Universal Robots PolyScope program: Aufgabe1_2.urp

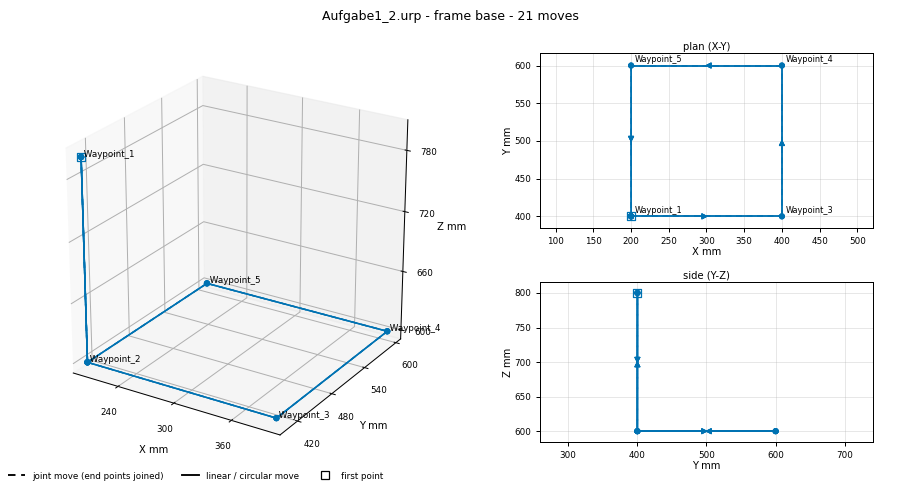
[picture p0: tool path of Aufgabe1_2.urp in frame base, 21 of 21 moves have a stored position in this frame; points joined in program order, loops and branches not executed]
Program Aufgabe1_2 (installation=default directory=/home/ur/ursim-current/programs/new folder createdIn=5.12.4.1101661 lastSavedIn=5.12.4.1101661 robotSerialNumber=20195599999)
Calibrated DH parameters: a=[0, -0.425, -0.3922, 0, 0, 0]; d=[0.1625, 0, 0, 0.1333, 0.0997, 0.0996]; alpha=[1.570796, 0, 0, 1.570796, -1.570796, 0]; deltaTheta=[0, 0, 0, 0, 0, 0]
Robot Program (runOnlyOnce=false)
  MoveL speed 250 mm/s, acceleration 1200 mm/s^2 (useActiveTCP=true) feature=Base
    Waypoint Waypoint_1: TCP in base x=200.031 y=400.097 z=800.02 mm, rx=0 ry=3.1204 rz=0 rad; joints [-133.696, -75.689, 20.033, -35.183, 269.122, 136.298] deg
    MoveL speed 250 mm/s, acceleration 1200 mm/s^2 (useActiveTCP=true) feature=Base
      Waypoint Waypoint_2: TCP in base x=200.014 y=400.002 z=600.007 mm, rx=0 ry=3.1204 rz=0 rad; joints [-133.703, -96.648, 79.829, -74.02, 269.122, 136.29] deg
      Waypoint Waypoint_3: TCP in base x=400.007 y=400.002 z=600.007 mm, rx=0 ry=3.1204 rz=0 rad; joints [-148.515, -79.953, 62.627, -73.709, 269.366, 121.479] deg
      Waypoint Waypoint_4: TCP in base x=400.007 y=600.024 z=600.007 mm, rx=0 ry=3.1204 rz=0 rad; joints [-134.219, -48.622, 15.08, -57.305, 269.13, 135.774] deg
      Waypoint Waypoint_5: TCP in base x=200.031 y=600.024 z=600.007 mm, rx=0 ry=3.1204 rz=0 rad; joints [-120.435, -69.177, 48.455, -69.893, 268.953, 149.559] deg
      Waypoint Waypoint_2: TCP in base x=200.014 y=400.002 z=600.007 mm, rx=0 ry=3.1204 rz=0 rad; joints [-133.703, -96.648, 79.829, -74.02, 269.122, 136.29] deg
      MoveL speed 250 mm/s, acceleration 1200 mm/s^2 (useActiveTCP=true) feature=Base
        Waypoint Waypoint_1: TCP in base x=200.031 y=400.097 z=800.02 mm, rx=0 ry=3.1204 rz=0 rad; joints [-133.696, -75.689, 20.033, -35.183, 269.122, 136.298] deg
  MoveJ speed 60 deg/s, acceleration 80 deg/s^2 (useActiveTCP=true) feature=Base
    Waypoint Waypoint_1: TCP in base x=200.031 y=400.097 z=800.02 mm, rx=0 ry=3.1204 rz=0 rad; joints [-133.696, -75.689, 20.033, -35.183, 269.122, 136.298] deg
    MoveJ speed 60 deg/s, acceleration 80 deg/s^2 (useActiveTCP=true) feature=Base
      Waypoint Waypoint_2: TCP in base x=200.014 y=400.002 z=600.007 mm, rx=0 ry=3.1204 rz=0 rad; joints [-133.703, -96.648, 79.829, -74.02, 269.122, 136.29] deg
      Waypoint Waypoint_3: TCP in base x=400.007 y=400.002 z=600.007 mm, rx=0 ry=3.1204 rz=0 rad; joints [-148.515, -79.953, 62.627, -73.709, 269.366, 121.479] deg
      Waypoint Waypoint_4: TCP in base x=400.007 y=600.024 z=600.007 mm, rx=0 ry=3.1204 rz=0 rad; joints [-134.219, -48.622, 15.08, -57.305, 269.13, 135.774] deg
      Waypoint Waypoint_5: TCP in base x=200.031 y=600.024 z=600.007 mm, rx=0 ry=3.1204 rz=0 rad; joints [-120.435, -69.177, 48.455, -69.893, 268.953, 149.559] deg
      Waypoint Waypoint_2: TCP in base x=200.014 y=400.002 z=600.007 mm, rx=0 ry=3.1204 rz=0 rad; joints [-133.703, -96.648, 79.829, -74.02, 269.122, 136.29] deg
      MoveJ speed 60 deg/s, acceleration 80 deg/s^2 (useActiveTCP=true) feature=Base
        Waypoint Waypoint_1: TCP in base x=200.031 y=400.097 z=800.02 mm, rx=0 ry=3.1204 rz=0 rad; joints [-133.696, -75.689, 20.033, -35.183, 269.122, 136.298] deg
  MoveP speed 250 mm/s, acceleration 1200 mm/s^2 (blendRadius=0.025 useActiveTCP=true) feature=Base
    Waypoint Waypoint_1: TCP in base x=200.031 y=400.097 z=800.02 mm, rx=0 ry=3.1204 rz=0 rad; joints [-133.696, -75.689, 20.033, -35.183, 269.122, 136.298] deg
    MoveP speed 250 mm/s, acceleration 1200 mm/s^2 (blendRadius=0.025 useActiveTCP=true) feature=Base
      Waypoint Waypoint_2: TCP in base x=200.014 y=400.002 z=600.007 mm, rx=0 ry=3.1204 rz=0 rad; joints [-133.703, -96.648, 79.829, -74.02, 269.122, 136.29] deg
      Waypoint Waypoint_3: TCP in base x=400.007 y=400.002 z=600.007 mm, rx=0 ry=3.1204 rz=0 rad; joints [-148.515, -79.953, 62.627, -73.709, 269.366, 121.479] deg
      Waypoint Waypoint_4: TCP in base x=400.007 y=600.024 z=600.007 mm, rx=0 ry=3.1204 rz=0 rad; joints [-134.219, -48.622, 15.08, -57.305, 269.13, 135.774] deg
      Waypoint Waypoint_5: TCP in base x=200.031 y=600.024 z=600.007 mm, rx=0 ry=3.1204 rz=0 rad; joints [-120.435, -69.177, 48.455, -69.893, 268.953, 149.559] deg
      Waypoint Waypoint_2: TCP in base x=200.014 y=400.002 z=600.007 mm, rx=0 ry=3.1204 rz=0 rad; joints [-133.703, -96.648, 79.829, -74.02, 269.122, 136.29] deg
      MoveP speed 250 mm/s, acceleration 1200 mm/s^2 (blendRadius=0.025 useActiveTCP=true) feature=Base
        Waypoint Waypoint_1: TCP in base x=200.031 y=400.097 z=800.02 mm, rx=0 ry=3.1204 rz=0 rad; joints [-133.696, -75.689, 20.033, -35.183, 269.122, 136.298] deg
